FUNCTION Convert_BOOL_TO_WORD : BOOL
VAR_INPUT
	in : BOOL;
	out : REFERENCE TO WORD;
END_VAR
VAR
	converted : WORD;
END_VAR

converted := BOOL_TO_WORD(in);

IF (WORD_TO_BOOL(converted) <> in) THEN
	RETURN;
END_IF

out := converted;
Convert_BOOL_TO_WORD := TRUE;

END_FUNCTION

(* stored: Version 1.1.0.1, ProductVersion 3.1.4024.12
   POU Convert_BOOL_TO_WORD: Id {40421e94-96a2-47a4-ab2b-fa36addcf979}, SpecialFunc None *)
